// TIA Portal V16 export
// export: Created 2021-05-26T11:33:15.9964349Z, ExportSetting WithDefaults, DisplayName Totally Integrated Automation Portal, DisplayVersion V16 Update 4, DisplayName TIA Portal Version Control Interface, DisplayVersion V16 Update 2, DisplayName TIA Portal Openness, DisplayVersion V16 Update 4, DisplayName STEP 7 Professional, DisplayVersion V16 Update 4, DisplayName STEP 7 Safety, DisplayVersion V16, DisplayName WinCC Advanced, DisplayVersion V16 Update 4
ORGANIZATION_BLOCK "Cyclic_fastBC"   // OB30, LAD, CyclicInterrupt
{ S7_Optimized_Access := 'TRUE' }
VERSION : 0.1
// Project:   CRE-331M  SSA PLC control system
// Copyright: 2019 Cryoelectra GmbH
// Purpose:fast Communication between basecontroller and PLC
// Versions:  
// 0.0  26-Nov-2019  fam  initial version                                     00
// 0.1  16-Jun-2020   fam  changed doc V1_6                            01
// 0.2  14-Jul-2020    fam   changed doc V1_9                           02
// 0.3   20-Jul-2020   fam   changed doc V2_0                           03
// 0.4   23-Jul-2020   bam  changed Pin, Prdrv1,2 calc.            04
// 0.5   03-Aug-2020 fam  changed DSL Doc V1_7                   05
// 0.6   31-Aug-2020 fam  chnaged DLS doc V1_9                   06
// stored: AutoNumber true, IsIECCheckEnabled false, SetENOAutomatically false
   VAR_INPUT
      Initial_Call : Bool;   // Initial call of this OB
      Event_Count : Int;   // Events discarded
   END_VAR
   VAR_TEMP
      RETVAL_BC : Int;
      PwrReal : Real;
   END_VAR
BEGIN

NETWORK
TITLE = 
      AN    "COMM_UDP_DB".TSND_BC.Start;
      =     "COMM_UDP_DB".TSND_BC.Start;
      AN    "COMM_UDP_DB".TSND_BC.Start;
      =     "COMM_UDP_DB".TRCV1_BC.Start;


REGION Network 2: Send UDP package to BaseCon
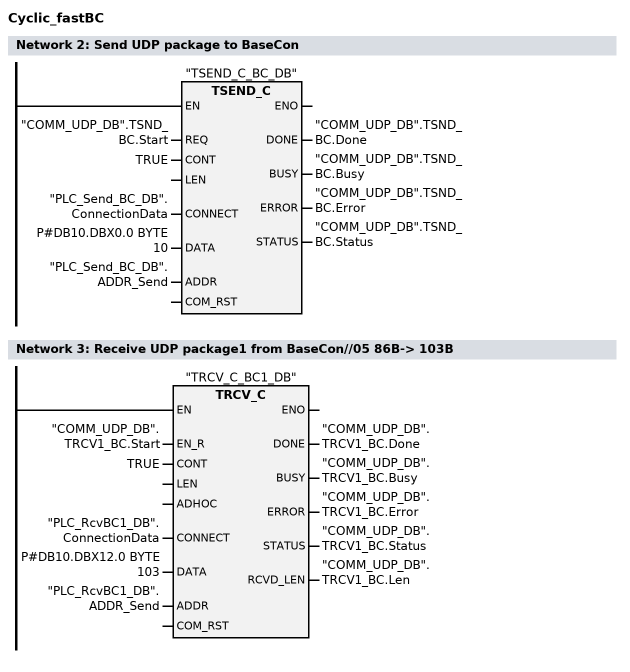
   RUNG wire#powerrail
      "TSEND_C_BC_DB".TSEND_C(REQ := "COMM_UDP_DB".TSND_BC.Start, CONT := TRUE, LEN :=, CONNECT := "PLC_Send_BC_DB".ConnectionData, DATA := P#DB10.DBX0.0 BYTE 10, ADDR := "PLC_Send_BC_DB".ADDR_Send, COM_RST :=, DONE => "COMM_UDP_DB".TSND_BC.Done, BUSY => "COMM_UDP_DB".TSND_BC.Busy, ERROR => "COMM_UDP_DB".TSND_BC.Error, STATUS => "COMM_UDP_DB".TSND_BC.Status)
   END_RUNG
   // the same network as SCL:
   "TSEND_C_BC_DB"(REQ := "COMM_UDP_DB".TSND_BC.Start,   // TSEND_C
                   CONT := TRUE,
                   CONNECT := "PLC_Send_BC_DB".ConnectionData,
                   DATA := P#DB10.DBX0.0 BYTE 10,
                   ADDR := "PLC_Send_BC_DB".ADDR_Send,
                   DONE => "COMM_UDP_DB".TSND_BC.Done,
                   BUSY => "COMM_UDP_DB".TSND_BC.Busy,
                   ERROR => "COMM_UDP_DB".TSND_BC.Error,
                   STATUS => "COMM_UDP_DB".TSND_BC.Status);
END_REGION

REGION Network 3: Receive UDP package1 from BaseCon//05 86B-> 103B
   RUNG wire#powerrail
      "TRCV_C_BC1_DB".TRCV_C(EN_R := "COMM_UDP_DB".TRCV1_BC.Start, CONT := TRUE, LEN :=, ADHOC :=, CONNECT := "PLC_RcvBC1_DB".ConnectionData, DATA := P#DB10.DBX12.0 BYTE 103, ADDR := "PLC_RcvBC1_DB".ADDR_Send, COM_RST :=, DONE => "COMM_UDP_DB".TRCV1_BC.Done, BUSY => "COMM_UDP_DB".TRCV1_BC.Busy, ERROR => "COMM_UDP_DB".TRCV1_BC.Error, STATUS => "COMM_UDP_DB".TRCV1_BC.Status, RCVD_LEN => "COMM_UDP_DB".TRCV1_BC.Len)
   END_RUNG
   // the same network as SCL:
   "TRCV_C_BC1_DB"(EN_R := "COMM_UDP_DB".TRCV1_BC.Start,   // TRCV_C
                   CONT := TRUE,
                   CONNECT := "PLC_RcvBC1_DB".ConnectionData,
                   DATA := P#DB10.DBX12.0 BYTE 103,
                   ADDR := "PLC_RcvBC1_DB".ADDR_Send,
                   DONE => "COMM_UDP_DB".TRCV1_BC.Done,
                   BUSY => "COMM_UDP_DB".TRCV1_BC.Busy,
                   ERROR => "COMM_UDP_DB".TRCV1_BC.Error,
                   STATUS => "COMM_UDP_DB".TRCV1_BC.Status,
                   RCVD_LEN => "COMM_UDP_DB".TRCV1_BC.Len);
END_REGION

NETWORK
TITLE = Received pacakge handling//06 05 01
      CALL  BLKMOV
      ( SRCBLK  := P#DB10.DBX12.0 BYTE 6,  //BYTE 6 10
        RET_VAL := #RETVAL_BC,
        DSTBLK  := P#DB70.DBX239.0 BYTE 6  //06 235
      );

      L     %DB10.DBW18;
      T     %DB70.DBW247;  //06 243
      L     %DB10.DBW20;
      T     %DB70.DBW245;  //06 241

      L     %DB10.DBB22;
      T     %DB70.DBB249;  //06 245

      L     "DB_BC".SW_Version;
      T     "DB_LPC".µCver_BC;



NETWORK
TITLE = Forward and Reflected Power calculations//05 03
      CALL  "FC_calcPwrFrwBC"
      ( Quell_DB     := "DB_BC",
        Quell_Offset := 38,  //05 36 PfrwMod1 in DB_BC
        Ziel_DB      := "DB_LPC",
        Ziel_Offset  := 78,  //06 74 CalPwrFrwMod1 in DB_LPC
        Anzahl       := 15
      );

      CALL  "FC_calcPwrRflBC"
      ( Quell_DB     := "DB_BC",
        Quell_Offset := 68,  //05 03 66 PrflMod1 in DB_BC
        Ziel_DB      := "DB_LPC",
        Ziel_Offset  := 142,  //06 138 CalPwrRflMod1
        Anzahl       := 15
      );

      CALL  "FC_eqPowerBC"
      ( P_Input   := "DB_BC".PwrFrwSsa,
        Cal_Param := "DB_LPC".calPwrFrwSSA,
        Ret_Val   := "DB_LPC".PwrFrwSsa
      );

      CALL  "FC_eqPowerBC"
      ( P_Input   := "DB_BC".PwrRflSsa,
        Cal_Param := "DB_LPC".calPwrRflSSA,
        Ret_Val   := "DB_LPC".PwrRflSsa
      );

      CALL  "FC_eqPowerBC"
      ( P_Input   := "DB_BC".PwrFrwDrv,
        Cal_Param := "DB_LPC".calPwrFrwDrv,
        Ret_Val   := #PwrReal
      );
      L     #PwrReal;
      RND;
      T     "DB_LPC".PwrFrwDrv;
      CALL  "FC_eqPowerBC"
      ( P_Input   := "DB_BC".PwrRflDrv,
        Cal_Param := "DB_LPC".calPwrRflDrv,
        Ret_Val   := #PwrReal
      );

      L     #PwrReal;
      RND;
      T     "DB_LPC".PwrRflDrv;

      CALL  "FC_eqPowerBC"
      ( P_Input   := "DB_BC".PwrPinSsa,
        Cal_Param := "DB_LPC".calPwrPinSSA,
        Ret_Val   := #PwrReal
      );
      L     #PwrReal;
      L     1000000.0;  //04
      *R;  //04
      RND;
      T     "DB_LPC".PwrPinSsa;  // in µW umrechnen !!!

      CALL  "FC_eqPowerBC"
      ( P_Input   := "DB_BC".PwrFrwPrDrv1,
        Cal_Param := "DB_LPC".calPwrFrwPrDrv1,
        Ret_Val   := #PwrReal
      );
      L     #PwrReal;
      L     1000000.0;  //04
      *R;  //04
      RND;
      T     "DB_LPC".PwrFrwPrDrv1;  //in µW umrechnen!!!

      CALL  "FC_eqPowerBC"
      ( P_Input   := "DB_BC".PwrFrwPrDrv2,
        Cal_Param := "DB_LPC".calPwrFrwPrDrv2,
        Ret_Val   := #PwrReal
      );
      L     #PwrReal;
      L     1000.0;  //04
      *R;  //04
      RND;
      T     "DB_LPC".PwrFrwPrDrv2;  //in mW umrechnen!!!
//05 added new data
      CALL  "FC_eqPowerBC"
      ( P_Input   := "DB_BC".PfrwCircIn,
        Cal_Param := "DB_LPC".calPfrwCircIn,
        Ret_Val   := "DB_LPC".PfrwCircIn
      );

      CALL  "FC_eqPowerBC"
      ( P_Input   := "DB_BC".PfrwCircOut,
        Cal_Param := "DB_LPC".calPfrwCircOut,
        Ret_Val   := "DB_LPC".PfrwCircOut
      );

      CALL  "FC_eqPowerBC"
      ( P_Input   := "DB_BC".PfrwCircLoad,
        Cal_Param := "DB_LPC".calPfrwCircLoad,
        Ret_Val   := "DB_LPC".PfrwCircLoad
      );

      CALL  "FC_eqPowerBC"
      ( P_Input   := "DB_BC".PfrwCoupl,
        Cal_Param := "DB_LPC".calPfrwCoupl,
        Ret_Val   := "DB_LPC".PfrwCoupl
      );

      CALL  "FC_eqPowerBC"
      ( P_Input   := "DB_BC".PrflCircIn,
        Cal_Param := "DB_LPC".calPrflCircIn,
        Ret_Val   := "DB_LPC".PrflCircIn
      );

      CALL  "FC_eqPowerBC"
      ( P_Input   := "DB_BC".PrflCircOut,
        Cal_Param := "DB_LPC".calPrflCircOut,
        Ret_Val   := "DB_LPC".PrflCircOut
      );
      CALL  "FC_eqPowerBC"
      ( P_Input   := "DB_BC".PrflCircLoad,
        Cal_Param := "DB_LPC".calPrflCircLoad,
        Ret_Val   := "DB_LPC".PrflCircLoad
      );
      CALL  "FC_eqPowerBC"
      ( P_Input   := "DB_BC".PrflCoupl,
        Cal_Param := "DB_LPC".calPrflCoupl,
        Ret_Val   := "DB_LPC".PrflCoupl
      );

















END_ORGANIZATION_BLOCK
